// TIA Portal project "ProjectCool" (V16)

(* hardware
DEVICE "S7300/ET200M station_1"  S7-300 station
   slot 0: "Rail_0"  Rail  6ES7 390-1***0-0AA0
   slot 2: "PLC_1"  CPU 314C-2 DP  6ES7 314-6CG03-0AB0  V2.6
      slot 0: "MPI interface_1"  X1
      slot 1: "DP interface_1"  X2
      slot 2: "DI 24/DO 16_1"  DI24/DO16
      slot 3: "AI 5/AO 2_1"  AI5/AO2
      slot 4: "Count_1"  Counter
      slot 5: "Positioning_1"  Positioning
   slot 4: "CP 343-1_1"  CP 343-1  6GK7 343-1EX11-0XE0  V2.0
*)

// ===== PLC "PLC_1"  CPU 314C-2 DP =====

VAR_GLOBAL   // PLC tag table "Default tag table"
   "Al3 - Masura" AT %IW6 : Int;
   "Ao0 - Comanda" AT %QW0 : Word;
   "Reset Bit" AT %M10.0 : Bool;
   "Referinta" AT %MD12 : Real;
   "AI1" AT %IW102 : Int;
END_VAR

DATA_BLOCK "data"   // DB1
{ S7_Optimized_Access := 'FALSE' }
VERSION : 0.1
   VAR
      "step" : Array[0..2000] of Real;
      data : Array[0..2000] of Real;
      index : Int;
      step_sample : Int;
      sample : Int;
   END_VAR
BEGIN
END_DATA_BLOCK

FUNCTION "mcc_data" : Void   // FC1, SCL
{ S7_Optimized_Access := 'FALSE' }
VERSION : 0.1
   VAR_INPUT
      initial_step : Real;   // initial step
      final_step : Real;   // final step
      step_time : Int;   // step time in ms
      sampling_time : Int;   // sampling time in ms
      step_period : Int;   // step period in ms
      PV : Int;   // process values
      Reset : Bool;   // reset aquisition procedure
   END_VAR
   VAR_OUTPUT
      MV : Word;   // manipulated value
   END_VAR
   VAR_TEMP
      ind : Int;   // actual sample
      index : Int;   // total number samples
      aux : Int;   // auxiliary variable
   END_VAR
   VAR CONSTANT
      n : Int := 2000;
   END_VAR
BEGIN
   #index := "data".index;
   IF (#index = 0) THEN
       "data".step_sample := #step_time / #sampling_time;
       "data".sample := #step_period / #sampling_time;
   END_IF;
   #ind := 0;
   IF (NOT #Reset AND #index < "data".step_sample) THEN
       #aux := REAL_TO_INT(#initial_step * 276.48);
       #MV := INT_TO_WORD(#aux);
   END_IF;
   IF (NOT #Reset AND #index <> -1 AND #index >= "data".step_sample AND #index < "data".step_sample + "data".sample) THEN
       #aux := REAL_TO_INT(#final_step * 276.48);
       #MV := INT_TO_WORD(#aux);
       #ind := #index - "data".step_sample + 1;
       "data".step[#ind] := #final_step - #initial_step;
       "data".data[#ind] := INT_TO_REAL(#PV) * 100 / 27648;
   END_IF;
   IF (NOT #Reset AND #index <> -1 AND #index < #n) THEN
       "data".index := #index + 1;
   ELSE
       "data".index := -1;
   END_IF;
   IF #Reset THEN
       "data".index := 0;
   END_IF;
END_FUNCTION

ORGANIZATION_BLOCK "Main"   // OB1, LAD
TITLE = "Main Program Sweep (Cycle)"
{ S7_Optimized_Access := 'FALSE' }
VERSION : 0.1
   VAR_TEMP
      OB1_EV_CLASS : Byte;   // Bits 0-3 = 1 (Coming event), Bits 4-7 = 1 (Event class 1)
      OB1_SCAN_1 : Byte;   // 1 (Cold restart scan 1 of OB 1), 3 (Scan 2-n of OB 1)
      OB1_PRIORITY : Byte;   // Priority of OB Execution
      OB1_OB_NUMBR : Byte;   // 1 (Organization block 1, OB1)
      OB1_RESERVED_1 : Byte;   // Reserved for system
      OB1_RESERVED_2 : Byte;   // Reserved for system
      OB1_PREV_CYCLE : Int;   // Cycle time of previous OB1 scan (milliseconds)
      OB1_MIN_CYCLE : Int;   // Minimum cycle time of OB1 (milliseconds)
      OB1_MAX_CYCLE : Int;   // Maximum cycle time of OB1 (milliseconds)
      OB1_DATE_TIME : Date_And_Time;   // Date and time OB1 started
   END_VAR
BEGIN
END_ORGANIZATION_BLOCK

ORGANIZATION_BLOCK "CYC_INT5"   // OB35, LAD
TITLE = "Cyclic Interrupt"
{ S7_Optimized_Access := 'FALSE' }
VERSION : 0.1
   VAR_TEMP
      OB35_EV_CLASS : Byte;   // Bits 0-3 = 1 (Coming event), Bits 4-7 = 1 (Event class 1)
      OB35_STRT_INF : Byte;   // 16#36 (OB 35 has started)
      OB35_PRIORITY : Byte;   // Priority of OB Execution
      OB35_OB_NUMBR : Byte;   // 35 (Organization block 35, OB35)
      OB35_RESERVED_1 : Byte;   // Reserved for system
      OB35_RESERVED_2 : Byte;   // Reserved for system
      OB35_PHASE_OFFSET : Word;   // Phase offset (msec)
      OB35_RESERVED_3 : Int;   // Reserved for system
      OB35_EXC_FREQ : Int;   // Frequency of execution (msec)
      OB35_DATE_TIME : Date_And_Time;   // Date and time OB35 started
   END_VAR
BEGIN

REGION Network 1
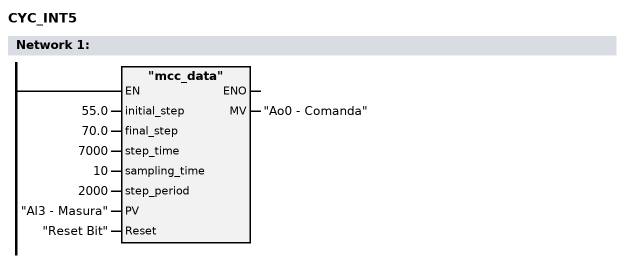
   RUNG wire#powerrail
      "mcc_data"(initial_step := 55.0, final_step := 70.0, step_time := 7000, sampling_time := 10, step_period := 2000, PV := "Al3 - Masura", Reset := "Reset Bit", MV => "Ao0 - Comanda")
   END_RUNG
   // the same network as SCL:
   "mcc_data"(initial_step := 55.0,
              final_step := 70.0,
              step_time := 7000,
              sampling_time := 10,
              step_period := 2000,
              PV := "Al3 - Masura",
              Reset := "Reset Bit",
              MV => "Ao0 - Comanda");
END_REGION
END_ORGANIZATION_BLOCK

ORGANIZATION_BLOCK "COMPLETE RESTART"   // OB100, SCL
TITLE = "Complete Restart"
{ S7_Optimized_Access := 'FALSE' }
VERSION : 0.1
   VAR_TEMP
      OB100_EV_CLASS : Byte;   // 16#13, Event class 1, Entering event state, Event logged in diagnostic buffer
      OB100_STRTUP : Byte;   // 16#81/82/83/84 Method of startup
      OB100_PRIORITY : Byte;   // Priority of OB Execution
      OB100_OB_NUMBR : Byte;   // 100 (Organization block 100, OB100)
      OB100_RESERVED_1 : Byte;   // Reserved for system
      OB100_RESERVED_2 : Byte;   // Reserved for system
      OB100_STOP : Word;   // Event that caused CPU to stop (16#4xxx)
      OB100_STRT_INFO : DWord;   // Information on how system started
      OB100_DATE_TIME : Date_And_Time;   // Date and time OB100 started
   END_VAR
BEGIN
   "data".index := 0;
END_ORGANIZATION_BLOCK